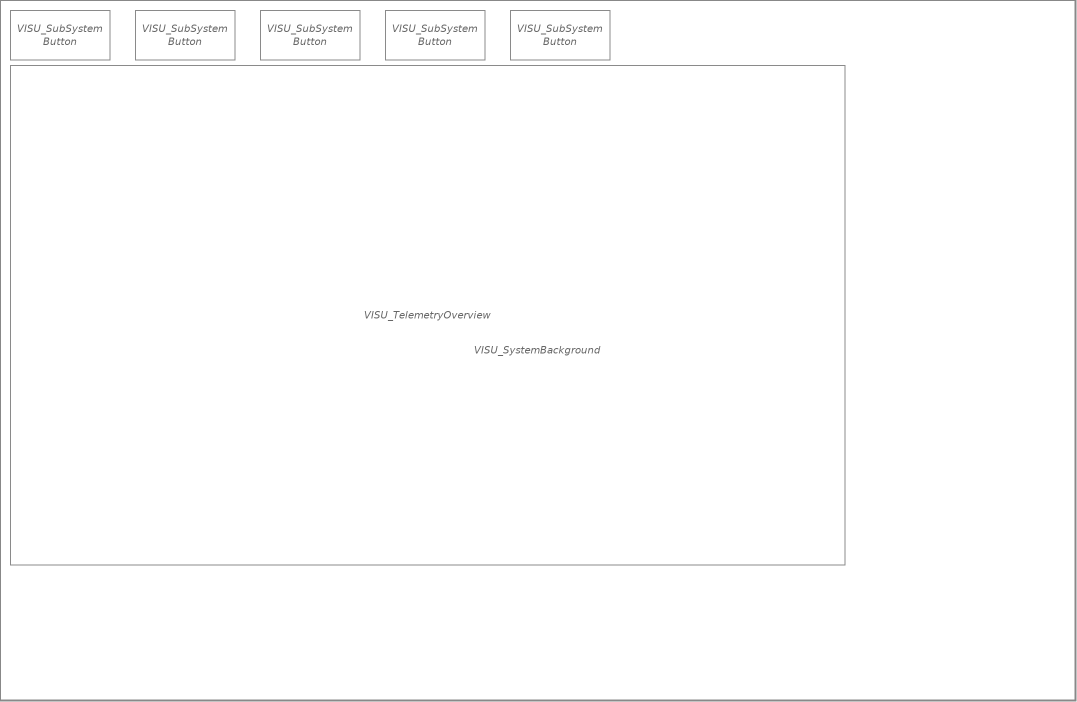
VISUALIZATION VISU_Telemetry  // 1077x702
VAR_IN_OUT
	ref : Telemetry;
    widget : TelemetryWidget;
END_VAR
    Frame (0,0 1075x700)
        shows VISU_SystemBackground(color := widget.actualStatus.color)
    Frame (10,65 835x500)
        shows VISU_TelemetryOverview(ref := ref, widget := widget)
        shows VISU_TelemetryFlatfieldLeds(ref := ref.parts.flatfieldLeds, widget := widget.flatfieldLeds)
        shows VISU_TelemetryAccelerometers(ref := ref.parts.accelerometers, widget := widget.accelerometers)
        shows VISU_TelemetryIO(ref := ref.parts.io, widget := widget.io)
        shows VISU_TelemetryConfig(editable := ref.editableConfig, active := ref.config, mgr := ref.parts.configManager, mgrWidget := widget.configManager, telemetryWidget := widget)
        p701045219: ref.editableConfig
        p2690442461: ref.config
        p942769723: ref.parts.configManager
        p2963374678: widget.configManager
        p459268616: widget
        p2421092570: ref.editableConfig
        p1485929088: ref.config
        p4084028830: ref.parts.configManager
        p721735225: widget.configManager
        p4094514409: widget
    Frame (10,10 100x50)
        shows VISU_SubSystemButton(widget := widget.button_overview)
        OnMouseClick: FrameSelectionChange Selection=SelectedFrame=b1e9e4b0-bf3d-440f-90c5-cb513105ccf1, GlobSel=AssignType=Directly, SelType=Locally
        OnMouseClick: execute { widget.activeTab := TelemetryTabs.OVERVIEW; }
    Frame (135,10 100x50)
        shows VISU_SubSystemButton(widget := widget.button_leds)
        OnMouseClick: FrameSelectionChange Selection=SelectedFrame=b1e9e4b0-bf3d-440f-90c5-cb513105ccf1, Selection=1, GlobSel=AssignType=Directly, SelType=Locally
        OnMouseClick: execute { widget.activeTab := TelemetryTabs.LEDS; }
    Frame (385,10 100x50)
        shows VISU_SubSystemButton(widget := widget.button_io)
        OnMouseClick: FrameSelectionChange Selection=SelectedFrame=b1e9e4b0-bf3d-440f-90c5-cb513105ccf1, Selection=3, GlobSel=AssignType=Directly, SelType=Locally
        OnMouseClick: execute { widget.activeTab := TelemetryTabs.IO; }
    Frame (510,10 100x50)
        shows VISU_SubSystemButton(widget := widget.button_config)
        OnMouseClick: FrameSelectionChange Selection=SelectedFrame=b1e9e4b0-bf3d-440f-90c5-cb513105ccf1, Selection=4, GlobSel=AssignType=Directly, SelType=Locally
        OnMouseClick: execute { widget.activeTab := TelemetryTabs.CONFIG; }
    Frame (260,10 100x50)
        shows VISU_SubSystemButton(widget := widget.button_accelerometers)
        OnMouseClick: FrameSelectionChange Selection=SelectedFrame=b1e9e4b0-bf3d-440f-90c5-cb513105ccf1, Selection=2, GlobSel=AssignType=Directly, SelType=Locally
        OnMouseClick: execute { widget.activeTab := TelemetryTabs.ACCELEROMETERS; }
END_VISUALIZATION

(* stored: Version 1.1.0.1, ProductVersion 3.1.4019.2
   Visu VISU_Telemetry: Id {58038c8c-ef69-4f6a-ae51-1c8458703a20} *)
